// TIA Portal V20 export
// export: Created 2026-07-30T13:06:46.5837966Z, ExportSetting WithDefaults, DisplayName Totally Integrated Automation Portal, DisplayVersion V20, DisplayName TIA Portal Openness, DisplayVersion V20, DisplayName TIA Portal Version Control Interface, DisplayVersion V20, DisplayName STEP 7 Professional, DisplayVersion V20, DisplayName STEP 7 Safety, DisplayVersion V20, DisplayName WinCC Basic/Comfort/Advanced, DisplayVersion V20, DisplayName WinCC Professional, DisplayVersion V20, DisplayName WinCC Unified, DisplayVersion V20
FUNCTION_BLOCK "FB_ValveLogic"   // FB3, SCL
{ S7_Optimized_Access := 'TRUE' }
VERSION : 0.1
// stored: AutoNumber true, IsIECCheckEnabled false, IsRetainMemResEnabled false, MemoryReserve 100, SetENOAutomatically false, UDAEnableTagReadback false
   VAR_IN_OUT
      Valve : "Valve_IO";
   END_VAR
BEGIN
   IF #Valve.Configured THEN

       // Mutual exclusion — Close takes priority if both are somehow TRUE
       IF #Valve.CloseCmd THEN
           #Valve.OpenCmd := FALSE;
       END_IF;
       IF #Valve.OpenCmd THEN
           #Valve.CloseCmd := FALSE;
       END_IF;

       // OPEN side
       IF #Valve.OpenCmd AND NOT #Valve.LocalMode AND #Valve.Healthy THEN
           #Valve.OpenValve := TRUE;
       ELSE
           #Valve.OpenValve := FALSE;
       END_IF;

       #Valve.TimerOpen(IN := #Valve.OpenValve,
                        PT := T#5s);
       IF #Valve.TimerOpen.Q THEN
           #Valve.OpenFB := TRUE;
           #Valve.ClosedFB := FALSE;
       END_IF;

       // CLOSE side
       IF #Valve.CloseCmd AND NOT #Valve.LocalMode AND #Valve.Healthy THEN
           #Valve.CloseValve := TRUE;
       ELSE
           #Valve.CloseValve := FALSE;
       END_IF;

       #Valve.TimerClose(IN := #Valve.CloseValve,
                         PT := T#5s);
       IF #Valve.TimerClose.Q THEN
           #Valve.ClosedFB := TRUE;
           #Valve.OpenFB := FALSE;
       END_IF;

   ELSE
       // Not configured — force everything safe/off
       #Valve.OpenValve := FALSE;
       #Valve.CloseValve := FALSE;
   END_IF;
END_FUNCTION_BLOCK
